// TIA Portal V17 export
// export: Created 2023-02-25T13:23:15.6641183Z, ExportSetting WithDefaults, DisplayName Totally Integrated Automation Portal, DisplayVersion V17, DisplayName TIA Portal Openness, DisplayVersion V17, DisplayName TIA Portal Version Control Interface, DisplayVersion V17, DisplayName TIA Portal Test Suite Advanced, DisplayVersion V17, DisplayName STEP 7 Professional, DisplayVersion V17, DisplayName SIMATIC Energy Suite, DisplayVersion V17, DisplayName STEP 7 Safety, DisplayVersion V17, DisplayName WinCC Professional, DisplayVersion V17
DATA_BLOCK "HW_MovingAverageFilter_DB"   // DB3
VERSION : 0.1
// stored: AutoNumber true, InstanceOfName HW_MovingAverageFilter, InstanceOfType FB
"HW_MovingAverageFilter"
   // VAR_INPUT
   //    Start : Bool;
   //    Samples : Int;
   //    Weight : Real;
   // END_VAR
   // VAR_OUTPUT
   //    WeightFilter : Real;
   // END_VAR
   // VAR
   //    Bufor : Array[0..99] of Real;
   // END_VAR
BEGIN
END_DATA_BLOCK
